KUKA KRL program: f_fraes4.src, f_fraes4.dat

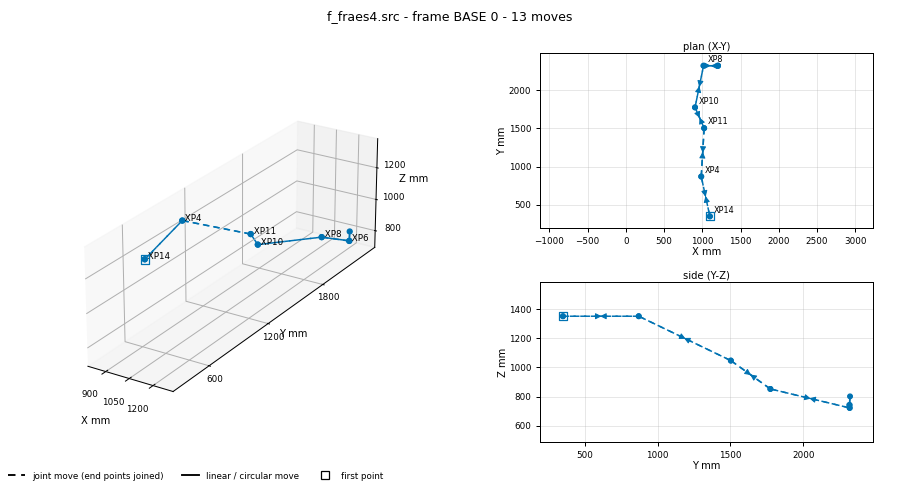
[picture p0: tool path of f_fraes4.src in frame BASE 0, 13 of 13 moves have a stored position in this frame; points joined in program order, loops and branches not executed]
--- f_fraes4.src ---
&ACCESS RVO7
&REL 23
&COMMENT INI Dress C3
&PARAM DISKPATH = KRC:\R1\Program
&PARAM TEMPLATE = C:\KRC\Roboter\Template\vorgabe
&PARAM EDITMASK = *
DEF f_fraes4( )
;FOLD INI
  ;FOLD BASISTECH INI
    GLOBAL INTERRUPT DECL 3 WHEN $STOPMESS==TRUE DO IR_STOPM ( )
    INTERRUPT ON 3
    BAS (#INITMOV,0 )
  ;ENDFOLD (BASISTECH INI)
;FOLD SPOTTECH INI
USERSPOT(#INIT)
;ENDFOLD (SPOTTECH INI)
;FOLD GRIPPERTECH INI
USER_GRP(0,DUMMY,DUMMY,GDEFAULT)
;ENDFOLD (GRIPPERTECH INI)
  ;FOLD USER INI
    ;Make your modifications here

  ;ENDFOLD (USER INI)
;ENDFOLD (INI)

; Caracterização dos meios de produção:
; Changes: Fresagem Final Gun C3
; Versão Atual:03/10/2015
; Name: P13.050-R1

chk_w4_wechs_ok() ; check c3


;FOLD PTP P14 CONT Vel=100 % PDAT24 Tool[4]:GUN C3 Base[0];%{PE}%R 8.2.20,%MKUKATPBASIS,%CMOVE,%VPTP,%P 1:PTP, 2:P14, 3:C_DIS, 5:100, 7:PDAT24
$BWDSTART=FALSE
PDAT_ACT=PPDAT24
FDAT_ACT=FP14
BAS(#PTP_PARAMS,100)
PTP XP14 C_DIS
;ENDFOLD
;FOLD PTP P4 CONT Vel=100 % PDAT12 Tool[4]:GUN C3 Base[0];%{PE}%R 8.2.20,%MKUKATPBASIS,%CMOVE,%VPTP,%P 1:PTP, 2:P4, 3:C_DIS, 5:100, 7:PDAT12
$BWDSTART=FALSE
PDAT_ACT=PPDAT12
FDAT_ACT=FP4
BAS(#PTP_PARAMS,100)
PTP XP4 C_DIS
;ENDFOLD
;FOLD PTP P11 CONT Vel=100 % PDAT21 Tool[4]:GUN C3 Base[0];%{PE}%R 8.2.20,%MKUKATPBASIS,%CMOVE,%VPTP,%P 1:PTP, 2:P11, 3:C_DIS, 5:100, 7:PDAT21
$BWDSTART=FALSE
PDAT_ACT=PPDAT21
FDAT_ACT=FP11
BAS(#PTP_PARAMS,100)
PTP XP11 C_DIS
;ENDFOLD
;FOLD PTP P10 CONT Vel=100 % PDAT20 Tool[4]:GUN C3 Base[0];%{PE}%R 8.2.20,%MKUKATPBASIS,%CMOVE,%VPTP,%P 1:PTP, 2:P10, 3:C_DIS, 5:100, 7:PDAT20
$BWDSTART=FALSE
PDAT_ACT=PPDAT20
FDAT_ACT=FP10
BAS(#PTP_PARAMS,100)
PTP XP10 C_DIS
;ENDFOLD
;FOLD PTP P8 CONT Vel=100 % PDAT18 Tool[4]:GUN C3 Base[0];%{PE}%R 8.2.20,%MKUKATPBASIS,%CMOVE,%VPTP,%P 1:PTP, 2:P8, 3:C_DIS, 5:100, 7:PDAT18
$BWDSTART=FALSE
PDAT_ACT=PPDAT18
FDAT_ACT=FP8
BAS(#PTP_PARAMS,100)
PTP XP8 C_DIS
;ENDFOLD

;FOLD LIN P6 Vel=1 m/s CPDAT4 Tool[4]:GUN C3 Base[0];%{PE}%R 8.2.20,%MKUKATPBASIS,%CMOVE,%VLIN,%P 1:LIN, 2:P6, 3:, 5:1, 7:CPDAT4
$BWDSTART=FALSE
LDAT_ACT=LCPDAT4
FDAT_ACT=FP6
BAS(#CP_PARAMS,1)
LIN XP6
;ENDFOLD

;FOLD ; PONTO DE FRESAGEM;%{PE}%R 8.2.20,%MKUKATPBASIS,%CCOMMENT,%VNORMAL,%P 2:PONTO  DE  FRESAGEM
;ENDFOLD
;FOLD TIP.PTP_ Dress4, Spot Gun 3 , RETR open , Tool[4], Base[0], EXT.TCP=FALSE;%{PE}%MKUKATPUSER
FDAT_ACT=FDress4
BAS(#FRAMES)
PTP  XDress4
S_ACT.GUN=3
S_ACT.RETR=#opn
S_READY=FALSE
USERSPOT (#DRESS,S_ACT )
WAIT FOR  S_READY
;ENDFOLD

;FOLD LIN P7 Vel=1 m/s CPDAT5 Tool[4]:GUN C3 Base[0];%{PE}%R 8.2.20,%MKUKATPBASIS,%CMOVE,%VLIN,%P 1:LIN, 2:P7, 3:, 5:1, 7:CPDAT5
$BWDSTART=FALSE
LDAT_ACT=LCPDAT5
FDAT_ACT=FP7
BAS(#CP_PARAMS,1)
LIN XP7
;ENDFOLD

;FOLD PTP p001 PDAT10 SPOT Gun=3 RETR OPN PgNo1=253 ACTIVE=1 Tool[4]:GUN C3 Base[0];%{PE}%R 8.2.2,%MKUKATPSPOT,%CSPOT,%VPTP,%P 1:PTP, 2:p001, 3:, 5:100, 7:PDAT10, 10:3, 12:#FIRST, 14:#OPN, 16:253, 18:1, 20:0, 22:0, 24:1, 25:NORMAL
$BWDSTART=FALSE
PDAT_ACT=PPDAT10
FDAT_ACT=Fp001
BAS(#PTP_PARAMS,PPDAT10.VEL)
S_ACT.GUN=3
S_ACT.PAIR=SDEFAULT.PAIR
S_ACT.RETR=#OPN
S_ACT.CLO_TM=1
S_ACT.PGNO1=253
S_ACT.PGNO2=SDEFAULT.PGNO2
S_ACT.PRESS1=SDEFAULT.PRESS1
S_ACT.PRESS2=SDEFAULT.PRESS2
S_READY=FALSE
PTP Xp001
USERSPOT(#SPOT, S_ACT)
WAIT FOR S_READY
;ENDFOLD
;FOLD PTP P9 CONT Vel=100 % PDAT19 Tool[4]:GUN C3 Base[0];%{PE}%R 8.2.20,%MKUKATPBASIS,%CMOVE,%VPTP,%P 1:PTP, 2:P9, 3:C_DIS, 5:100, 7:PDAT19
$BWDSTART=FALSE
PDAT_ACT=PPDAT19
FDAT_ACT=FP9
BAS(#PTP_PARAMS,100)
PTP XP9 C_DIS
;ENDFOLD
;FOLD PTP P12 CONT Vel=100 % PDAT22 Tool[4]:GUN C3 Base[0];%{PE}%R 8.2.20,%MKUKATPBASIS,%CMOVE,%VPTP,%P 1:PTP, 2:P12, 3:C_DIS, 5:100, 7:PDAT22
$BWDSTART=FALSE
PDAT_ACT=PPDAT22
FDAT_ACT=FP12
BAS(#PTP_PARAMS,100)
PTP XP12 C_DIS
;ENDFOLD
;FOLD PTP P13 CONT Vel=100 % PDAT23 Tool[4]:GUN C3 Base[0];%{PE}%R 8.2.20,%MKUKATPBASIS,%CMOVE,%VPTP,%P 1:PTP, 2:P13, 3:C_DIS, 5:100, 7:PDAT23
$BWDSTART=FALSE
PDAT_ACT=PPDAT23
FDAT_ACT=FP13
BAS(#PTP_PARAMS,100)
PTP XP13 C_DIS
;ENDFOLD
;FOLD PTP P17 CONT Vel=100 % PDAT27 Tool[4]:GUN C3 Base[0];%{PE}%R 8.2.20,%MKUKATPBASIS,%CMOVE,%VPTP,%P 1:PTP, 2:P17, 3:C_DIS, 5:100, 7:PDAT27
$BWDSTART=FALSE
PDAT_ACT=PPDAT27
FDAT_ACT=FP17
BAS(#PTP_PARAMS,100)
PTP XP17 C_DIS
;ENDFOLD

END

--- f_fraes4.dat ---
&ACCESS RVO7
&REL 23
&COMMENT INI Dress C3
&PARAM DISKPATH = KRC:\R1\Program
&PARAM TEMPLATE = C:\KRC\Roboter\Template\vorgabe
&PARAM EDITMASK = *
DEFDAT  f_fraes4
;FOLD EXTERNAL DECLARATIONS;%{PE}%MKUKATPBASIS,%CEXT,%VCOMMON,%P
;FOLD GRIPPERTECH EXT
EXT  H50 (INT  :IN,INT  :IN,INT  :IN,GRP_TYP  :IN )
;ENDFOLD (GRIPPERTECH EXT)
;FOLD SPOTTECH EXT
EXT  USERSPOT (S_COMMAND  :IN,SPOT_TYPE  :IN )
;ENDFOLD (SPOTTECH EXT)
;FOLD BASISTECH EXT;%{PE}%MKUKATPBASIS,%CEXT,%VEXT,%P
EXT  BAS (BAS_COMMAND  :IN,REAL  :IN )
DECL INT SUCCESS
;ENDFOLD (BASISTECH EXT)
;FOLD USER EXT;%{E}%MKUKATPUSER,%CEXT,%VEXT,%P
;Make your modifications here

;ENDFOLD (USER EXT)
;ENDFOLD (EXTERNAL DECLARATIONS)
DECL BASIS_SUGG_T LAST_BASIS={POINT1[] "P17                     ",POINT2[] "P17                     ",CP_PARAMS[] "CPDAT3                  ",PTP_PARAMS[] "PDAT27                  ",CONT[] "C_DIS                   ",CP_VEL[] "1                       ",PTP_VEL[] "100                     ",SYNC_PARAMS[] "SYNCDAT                 ",SPL_NAME[] "S0                      "}
DECL SPOT_SUGG_T LAST_SPOT={GUN[] "4                       ",RETR_CMD[] "#OPN                    ",CHOISE[] "#FIRST                  ",CLO_TM[] "1                       ",PGNO1[] "1                       ",PRESS1[] "0                       ",PGNO2[] "1                       ",PRESS2[] "0                       ",SPOT_PARAMS[] "NORMAL                  "}
DECL PDAT PPDAT10={VEL 100.0,ACC 100.0,APO_DIST 100.0,APO_MODE #CDIS}
DECL E6POS Xp001={X 1016.30603,Y 2319.70508,Z 721.820374,A 1.503088,B -2.0431931,C 0.318278402,S 2,T 35,E1 383.111603,E2 0.0,E3 0.0,E4 0.0,E5 0.0,E6 0.0}
DECL FDAT Fp001={TOOL_NO 4,BASE_NO 0,IPO_FRAME #BASE,POINT2[] " ",TQ_STATE FALSE}
DECL E6POS XP4={X 986.087891,Y 869.488281,Z 1352.21301,A 27.6427708,B -8.47195053,C 0.388619512,S 2,T 11,E1 383.09201,E2 0.0,E3 0.0,E4 0.0,E5 0.0,E6 0.0}
DECL FDAT FP4={TOOL_NO 4,BASE_NO 0,IPO_FRAME #BASE,POINT2[] " ",TQ_STATE FALSE}
DECL PDAT PPDAT12={VEL 100.0,ACC 100.0,APO_DIST 200.0,APO_MODE #CDIS}
DECL FDAT FDress4={TOOL_NO 4,BASE_NO 0,IPO_FRAME #BASE}
DECL E6POS XDress4={X 1204.37805,Y 2322.13892,Z 801.162292,A -0.69191891,B -0.744428873,C -0.249322206,S 2,T 35,E1 383.095886,E2 0.0,E3 0.0,E4 0.0,E5 0.0,E6 0.0}
DECL E6POS XP6={X 1204.98303,Y 2319.68408,Z 742.008728,A 2.58857608,B -2.04355788,C 0.3180902,S 2,T 35,E1 383.111298,E2 0.0,E3 0.0,E4 0.0,E5 0.0,E6 0.0}
DECL FDAT FP6={TOOL_NO 4,BASE_NO 0,IPO_FRAME #BASE,POINT2[] " ",TQ_STATE FALSE}
DECL PDAT PPDAT16={VEL 100.0,ACC 100.0,APO_DIST 100.0,APO_MODE #CDIS}
DECL E6POS XP7={X 1204.98303,Y 2317.13696,Z 742.008728,A 1.503057,B -2.04319096,C 0.318306386,S 2,T 35,E1 383.111298,E2 0.0,E3 0.0,E4 0.0,E5 0.0,E6 0.0}
DECL FDAT FP7={TOOL_NO 4,BASE_NO 0,IPO_FRAME #BASE,POINT2[] " ",TQ_STATE FALSE}
DECL PDAT PPDAT17={VEL 100.0,ACC 100.0,APO_DIST 100.0,APO_MODE #CDIS}
DECL E6POS XP8={X 1016.30603,Y 2319.70508,Z 721.820374,A 1.503088,B -2.0431931,C 0.318278402,S 2,T 35,E1 383.111603,E2 0.0,E3 0.0,E4 0.0,E5 0.0,E6 0.0}
DECL FDAT FP8={TOOL_NO 4,BASE_NO 0,IPO_FRAME #BASE,POINT2[] " ",TQ_STATE FALSE}
DECL PDAT PPDAT18={VEL 100.0,ACC 100.0,APO_DIST 100.0,APO_MODE #CDIS}
DECL E6POS XP9={X 904.782776,Y 1774.49597,Z 852.132629,A 2.91674995,B -2.04276109,C 0.31771031,S 2,T 35,E1 383.111908,E2 0.0,E3 0.0,E4 0.0,E5 0.0,E6 0.0}
DECL FDAT FP9={TOOL_NO 4,BASE_NO 0,IPO_FRAME #BASE,POINT2[] " ",TQ_STATE FALSE}
DECL PDAT PPDAT19={VEL 100.0,ACC 100.0,APO_DIST 100.0,APO_MODE #CDIS}
DECL E6POS XP10={X 904.782776,Y 1774.49597,Z 852.132629,A 2.91674995,B -2.04276109,C 0.31771031,S 2,T 35,E1 383.111908,E2 0.0,E3 0.0,E4 0.0,E5 0.0,E6 0.0}
DECL FDAT FP10={TOOL_NO 4,BASE_NO 0,IPO_FRAME #BASE,POINT2[] " ",TQ_STATE FALSE}
DECL PDAT PPDAT20={VEL 100.0,ACC 100.0,APO_DIST 100.0,APO_MODE #CDIS}
DECL E6POS XP11={X 1024.22095,Y 1502.71301,Z 1047.18201,A 5.80271578,B -0.780567586,C 1.58314002,S 2,T 43,E1 383.116394,E2 0.0,E3 0.0,E4 0.0,E5 0.0,E6 0.0}
DECL FDAT FP11={TOOL_NO 4,BASE_NO 0,IPO_FRAME #BASE,POINT2[] " ",TQ_STATE FALSE}
DECL PDAT PPDAT21={VEL 100.0,ACC 100.0,APO_DIST 100.0,APO_MODE #CDIS}
DECL E6POS XP12={X 1024.22095,Y 1502.71301,Z 1047.18201,A 5.80271578,B -0.780567586,C 1.58314002,S 2,T 43,E1 383.116394,E2 0.0,E3 0.0,E4 0.0,E5 0.0,E6 0.0}
DECL FDAT FP12={TOOL_NO 4,BASE_NO 0,IPO_FRAME #BASE,POINT2[] " ",TQ_STATE FALSE}
DECL PDAT PPDAT22={VEL 100.0,ACC 100.0,APO_DIST 100.0,APO_MODE #CDIS}
DECL E6POS XP13={X 986.087891,Y 869.488281,Z 1352.21301,A 27.6427708,B -8.47195053,C 0.388619512,S 2,T 11,E1 383.09201,E2 0.0,E3 0.0,E4 0.0,E5 0.0,E6 0.0}
DECL FDAT FP13={TOOL_NO 4,BASE_NO 0,IPO_FRAME #BASE,POINT2[] " ",TQ_STATE FALSE}
DECL PDAT PPDAT23={VEL 100.0,ACC 100.0,APO_DIST 100.0,APO_MODE #CDIS}
DECL FDAT FDress6={TOOL_NO 4,BASE_NO 0,IPO_FRAME #BASE}
DECL E6POS XDress6={X 1207.35901,Y 2321.42993,Z 785.573486,A 1.50301003,B -2.04312205,C 0.318279088,S 2,T 35,E1 383.110413,E2 0.0,E3 0.0,E4 0.0,E5 0.0,E6 0.0}
DECL E6POS XP14={X 1098.979,Y 348.582001,Z 1352.20898,A -0.411624402,B -8.47158909,C 0.388728887,S 2,T 11,E1 383.0979,E2 0.0,E3 0.0,E4 0.0,E5 0.0,E6 0.0}
DECL FDAT FP14={TOOL_NO 4,BASE_NO 0,IPO_FRAME #BASE,POINT2[] " ",TQ_STATE FALSE}
DECL PDAT PPDAT24={VEL 100.0,ACC 100.0,APO_DIST 200.0,APO_MODE #CDIS}
DECL E6POS XP15={X 845.888611,Y -742.939819,Z 1352.21106,A -38.3194885,B -8.47178268,C 0.388727814,S 2,T 11,E1 -40.4965591,E2 0.0,E3 0.0,E4 0.0,E5 0.0,E6 0.0}
DECL FDAT FP15={TOOL_NO 4,BASE_NO 0,IPO_FRAME #BASE,POINT2[] " ",TQ_STATE FALSE}
DECL PDAT PPDAT25={VEL 100.0,ACC 100.0,APO_DIST 200.0,APO_MODE #CDIS}
DECL LDAT LCPDAT4={VEL 2.0,ACC 100.0,APO_DIST 100.0,APO_FAC 50.0,AXIS_VEL 100.0,AXIS_ACC 100.0,ORI_TYP #VAR,CIRC_TYP #BASE,JERK_FAC 50.0,GEAR_JERK 50.0,EXAX_IGN 0}
DECL LDAT LCPDAT5={VEL 2.0,ACC 100.0,APO_DIST 100.0,APO_FAC 50.0,AXIS_VEL 100.0,AXIS_ACC 100.0,ORI_TYP #VAR,CIRC_TYP #BASE,JERK_FAC 50.0,GEAR_JERK 50.0,EXAX_IGN 0}
DECL E6POS XP16={X 845.888611,Y -742.939819,Z 1352.21106,A -38.3194885,B -8.47178268,C 0.388727814,S 2,T 11,E1 -40.4965591,E2 0.0,E3 0.0,E4 0.0,E5 0.0,E6 0.0}
DECL FDAT FP16={TOOL_NO 4,BASE_NO 0,IPO_FRAME #BASE,POINT2[] " ",TQ_STATE FALSE}
DECL PDAT PPDAT26={VEL 100.0,ACC 100.0,APO_DIST 100.0,APO_MODE #CDIS}
DECL PDAT PPDAT27={VEL 100.0,ACC 100.0,APO_DIST 200.0,APO_MODE #CDIS}
DECL E6POS XP17={X 1098.979,Y 348.582001,Z 1352.20898,A -0.411624402,B -8.47158909,C 0.388728887,S 2,T 11,E1 383.0979,E2 0.0,E3 0.0,E4 0.0,E5 0.0,E6 0.0}
DECL FDAT FP17={TOOL_NO 4,BASE_NO 0,IPO_FRAME #BASE,POINT2[] " ",TQ_STATE FALSE}
ENDDAT
